TYPE ST_HexMove_Output :
STRUCT
	Disp_P: matrix_18_real_T;
END_STRUCT
END_TYPE

(* stored: Version 1.1.0.1, ProductVersion 3.1.4020.12
   DUT ST_HexMove_Output: Id {99954306-c44d-4c9f-9a56-8a1447a65979} *)
